FUNCTION_BLOCK HiveMQ_MQTT
VAR
	asd : FB_IotMqttClient := (sHostName := '5a4bc4b2d7c240d58dfbffe85ec21b83.s1.eu.hivemq.cloud');
	connect : BOOL := TRUE;
END_VAR

// asd(
// 	sClientId:= , 
// 	sHostName:= , 
// 	nHostPort:= , 
// 	sTopicPrefix:= , 
// 	nKeepAlive:= , 
// 	sUserName:= , 
// 	sUserPassword:= , 
// 	stWill:= , 
// 	stTLS:= , 
// 	ipMessageQueue:= , 
// 	bError=> , 
// 	hrErrorCode=> , 
// 	eConnectionState=> , 
// 	bConnected=> );
	
asd.Execute(connect);

METHOD CyclicCode
VAR_INPUT
END_VAR
END_METHOD

END_FUNCTION_BLOCK

(* stored: Version 1.1.0.1
   POU HiveMQ_MQTT: Id {cd48a2ab-b805-47d1-894a-d08367ff474b}, SpecialFunc None
   Method CyclicCode: Id {26710d21-e884-4fe8-8ad2-06fc4f639861} *)
